INTERFACE I_DataDisposer

METHOD DisposeData
VAR_INPUT
	Source : I_DataAccess;
END_VAR
END_METHOD

END_INTERFACE

(* stored: Version 1.1.0.1, ProductVersion 3.1.4024.12
   Itf I_DataDisposer: Id {4efb882e-a074-012a-0db9-6825328cb0ff}
   Method DisposeData: Id {9aa1e6b5-0262-094e-3ecb-e00254fe3512} *)
